// TIA Portal V18 export
FUNCTION_BLOCK "03_FDBACK error"   // FB4, F_LAD
{ S7_Optimized_Access := 'TRUE' }
   VAR_INPUT
      Commissioning_bypass : Bool;
      "FDBACK ERROR 1" : Bool;
      "FDBACK ERROR 2" : Bool;
      "FDBACK ERROR 3" : Bool;
      "FDBACK ERROR 4" : Bool;
      "FDBACK ERROR 5" : Bool;
      "FDBACK ERROR 6" : Bool;
      "FDBACK ERROR 7" : Bool;
      "FDBACK ERROR 8" : Bool;
   END_VAR
   VAR_OUTPUT
      "Cumulative FDBACK" : Bool;
      "ERROR 1" : Bool;
      "ERROR 2" : Bool;
      "ERROR 3" : Bool;
      "ERROR 4" : Bool;
      "ERROR 5" : Bool;
      "ERROR 6" : Bool;
      "ERROR 7" : Bool;
      "ERROR 8" : Bool;
   END_VAR
BEGIN

REGION Network 1: First channel
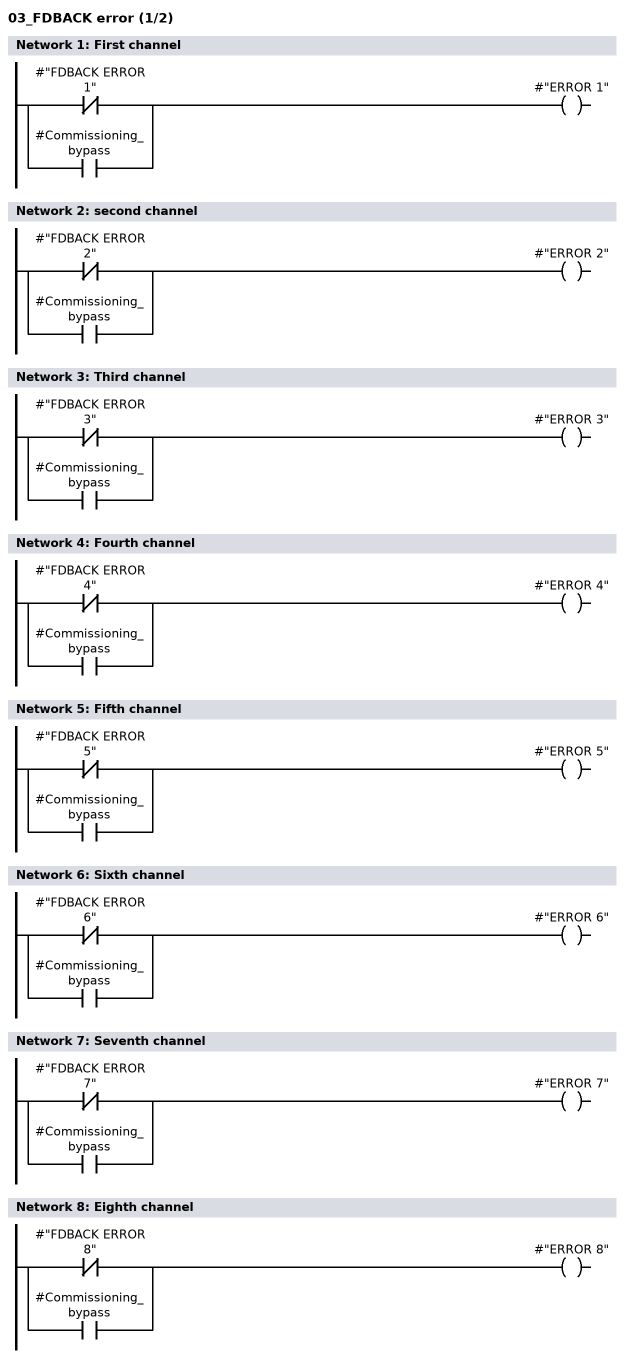
   RUNG wire#powerrail
      I_Contact( #"FDBACK ERROR 1" )
      wire#w1
      Coil( #"ERROR 1" )
   END_RUNG
   RUNG wire#powerrail
      Contact( #Commissioning_bypass )
   END_RUNG wire#w1
   // the same network as SCL:
   #"ERROR 1" := NOT #"FDBACK ERROR 1" OR #Commissioning_bypass;
END_REGION

REGION Network 2: second channel
   RUNG wire#powerrail
      I_Contact( #"FDBACK ERROR 2" )
      wire#w1
      Coil( #"ERROR 2" )
   END_RUNG
   RUNG wire#powerrail
      Contact( #Commissioning_bypass )
   END_RUNG wire#w1
   // the same network as SCL:
   #"ERROR 2" := NOT #"FDBACK ERROR 2" OR #Commissioning_bypass;
END_REGION

REGION Network 3: Third channel
   RUNG wire#powerrail
      I_Contact( #"FDBACK ERROR 3" )
      wire#w1
      Coil( #"ERROR 3" )
   END_RUNG
   RUNG wire#powerrail
      Contact( #Commissioning_bypass )
   END_RUNG wire#w1
   // the same network as SCL:
   #"ERROR 3" := NOT #"FDBACK ERROR 3" OR #Commissioning_bypass;
END_REGION

REGION Network 4: Fourth channel
   RUNG wire#powerrail
      I_Contact( #"FDBACK ERROR 4" )
      wire#w1
      Coil( #"ERROR 4" )
   END_RUNG
   RUNG wire#powerrail
      Contact( #Commissioning_bypass )
   END_RUNG wire#w1
   // the same network as SCL:
   #"ERROR 4" := NOT #"FDBACK ERROR 4" OR #Commissioning_bypass;
END_REGION

REGION Network 5: Fifth channel
   RUNG wire#powerrail
      I_Contact( #"FDBACK ERROR 5" )
      wire#w1
      Coil( #"ERROR 5" )
   END_RUNG
   RUNG wire#powerrail
      Contact( #Commissioning_bypass )
   END_RUNG wire#w1
   // the same network as SCL:
   #"ERROR 5" := NOT #"FDBACK ERROR 5" OR #Commissioning_bypass;
END_REGION

REGION Network 6: Sixth channel
   RUNG wire#powerrail
      I_Contact( #"FDBACK ERROR 6" )
      wire#w1
      Coil( #"ERROR 6" )
   END_RUNG
   RUNG wire#powerrail
      Contact( #Commissioning_bypass )
   END_RUNG wire#w1
   // the same network as SCL:
   #"ERROR 6" := NOT #"FDBACK ERROR 6" OR #Commissioning_bypass;
END_REGION

REGION Network 7: Seventh channel
   RUNG wire#powerrail
      I_Contact( #"FDBACK ERROR 7" )
      wire#w1
      Coil( #"ERROR 7" )
   END_RUNG
   RUNG wire#powerrail
      Contact( #Commissioning_bypass )
   END_RUNG wire#w1
   // the same network as SCL:
   #"ERROR 7" := NOT #"FDBACK ERROR 7" OR #Commissioning_bypass;
END_REGION

REGION Network 8: Eighth channel
   RUNG wire#powerrail
      I_Contact( #"FDBACK ERROR 8" )
      wire#w1
      Coil( #"ERROR 8" )
   END_RUNG
   RUNG wire#powerrail
      Contact( #Commissioning_bypass )
   END_RUNG wire#w1
   // the same network as SCL:
   #"ERROR 8" := NOT #"FDBACK ERROR 8" OR #Commissioning_bypass;
END_REGION

REGION Network 9: Cumulative error
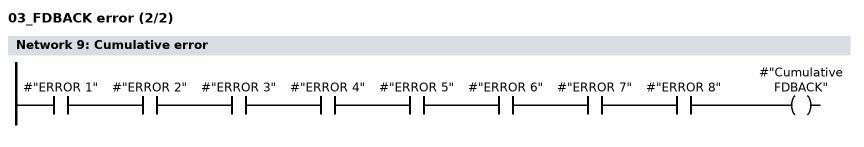
   RUNG wire#powerrail
      Contact( #"ERROR 1" )
      Contact( #"ERROR 2" )
      Contact( #"ERROR 3" )
      Contact( #"ERROR 4" )
      Contact( #"ERROR 5" )
      Contact( #"ERROR 6" )
      Contact( #"ERROR 7" )
      Contact( #"ERROR 8" )
      Coil( #"Cumulative FDBACK" )
   END_RUNG
   // the same network as SCL:
   #"Cumulative FDBACK" := #"ERROR 1" AND #"ERROR 2" AND #"ERROR 3" AND #"ERROR 4" AND #"ERROR 5" AND #"ERROR 6" AND #"ERROR 7" AND #"ERROR 8";
END_REGION
END_FUNCTION_BLOCK
